// TIA Portal V20 export
FUNCTION_BLOCK "FB_PowerOn"   // FB462, SCL
{ S7_Optimized_Access := 'TRUE' }
// stored: AutoNumber false, MemoryReserve 100, SetENOAutomatically false
   VAR
      sMachinePower : Bool;
      sMachineReadySoft : Bool;
      sOkForPowerON : Bool;
      sTimeMachineReadyDelay { S7_SetPoint := 'True'} : TON_TIME;
      sDelayPowerOFF { S7_SetPoint := 'True'} : TON_TIME;
      sDelayPowerON_1 { S7_SetPoint := 'True'} : TON_TIME;
      sDelayPowerON_2 { S7_SetPoint := 'True'} : TON_TIME;
      sX_AxisBrakeRelease { S7_SetPoint := 'True'} : Bool;
      sY_AxisBrakeRelease : Bool;
      sB_AxisBrakeRelease : Bool;
   END_VAR
   VAR CONSTANT
      TIME_MACHINE_IN_DELAY : Time := T#2S;   // Output short pulse blinking
   END_VAR
BEGIN
   REGION Description header 
       //==================================================================================
       // POSALUX Swiss SA / (C) Copyright 2024
       //----------------------------------------------------------------------------------
       // Title: Power de la machine
       // Comment/Function: 
       //  A revoir le power des differents elements
       // Author: Gowsigan SRITHARAN
       // Engineering: TIA Portal v17
       //----------------------------------------------------------------------------------
       // Change log table:
       // Version  | Date     | Expert in charge | Changes applied
       // ---------|----------|------------------|------------------------------------
       // 00.00.01 | 20241120 | GSR              | First released version
       // ==================================================================================
   END_REGION

   REGION General Circuit breaker
       IF NOT "DB_DigitalInputs".sBreakerCtrl.sSWStatus THEN
           "LBP_AlarmMsgs".UserA[0].A70UUxx[3] := TRUE;
       END_IF;
   END_REGION

   REGION Operating counter
       "DB_DigitalOutputs".sOperatingCounter.sSWStatus :=
       ("LBP_Chan1".E_ProgRunning
       OR "LBP_Chan1".E_ProgWait)
       AND "LBP_ModeGroup".E_AUTO;
   END_REGION

   REGION Axis power requested
       #sOkForPowerON := "LBP_NC".E_NCKready AND "LBP_NC".E_DrivesInCylOp AND "DB_DataFromSafety".EmergencyStop AND NOT "DB_Alarms".sAlarmsLevel5 AND NOT "DB_Alarms".sAlarmsLevel6;

       IF #sOkForPowerON AND "DB_McpKeyboardSignals".sPowerON.sKeySWPositiveFront THEN
           #sMachinePower := TRUE;
       END_IF;

       IF  "DB_McpKeyboardSignals".sPowerOFF.sKeySWNegativeFront
           OR "DB_Machineshutdown_UPS".sShutDownPower
           OR "DB_Alarms".sAlarmsLevel5
           OR NOT "DB_DataFromSafety".EmergencyStop THEN
           #sMachinePower := FALSE;
       END_IF;

   END_REGION

   REGION Axis power output and waiting machine ready
       #sDelayPowerOFF(IN := NOT "LBP_NC".E_611Dready AND NOT #sMachinePower,
                       PT := T#1s);

       #sDelayPowerON_1(IN := "DB_DigitalOutputs".sInfeedON.sSWStatus,
                        PT := t#2s);
       #sDelayPowerON_2(IN := "DB_DigitalOutputs".sAxisActivation.sSWStatus,
                        PT := t#2s);
       IF #sMachinePower THEN
           "DB_DigitalOutputs".sInfeedON.sSWStatus := TRUE;
           IF #sDelayPowerON_1.Q THEN
               "DB_DigitalOutputs".sAxisActivation.sSWStatus := TRUE;
           END_IF;
           IF #sDelayPowerON_2.Q THEN

               "DB_DigitalOutputs".sAxis2_PowerContactor.sSWStatus  := TRUE;
               "DB_DigitalOutputs".sXY_AxisPowerContactor.sSWStatus := TRUE;
               "DB_DigitalOutputs".sBus60V_PowerContactor.sSWStatus := TRUE;
           END_IF;
       ELSE
           "DB_DigitalOutputs".sAxisActivation.sSWStatus := FALSE;

           IF #sDelayPowerOFF.Q THEN
               "DB_DigitalOutputs".sAxis2_PowerContactor.sSWStatus  := FALSE;
               "DB_DigitalOutputs".sXY_AxisPowerContactor.sSWStatus := FALSE;
               "DB_DigitalOutputs".sBus60V_PowerContactor.sSWStatus := FALSE;
               "DB_DigitalOutputs".sInfeedON.sSWStatus := FALSE;
           END_IF;
       END_IF;

       #sMachineReadySoft := "LBP_NC".E_611Dready;
   END_REGION

   REGION Machine in delay
       #sTimeMachineReadyDelay.TON(IN := #sMachineReadySoft,
                                   PT := #TIME_MACHINE_IN_DELAY);
   END_REGION

   REGION LED Machine ready start
       "DB_McpKeyboardSignals".sPowerON.sLedSWStatus :=
       (NOT #sMachinePower AND #sOkForPowerON AND "Clock_0.5Hz")
       OR (NOT #sTimeMachineReadyDelay.Q AND #sMachinePower AND "Clock_2Hz")
       OR #sTimeMachineReadyDelay.Q AND #sMachineReadySoft;
   END_REGION

   REGION Axis Brake
       // X Axis Brake Activation
       "DB_DigitalOutputs".sX_AxisBrakeActivation.sSWStatus := (("LBP_Axis01_X".E_AxisReady
       AND "LBP_Axis01_X".E_MotOK
       AND "LBP_Axis01_X".E_PulseEnable)
       OR #sX_AxisBrakeRelease);

       // Y Axis Brake Activation    
       "DB_DigitalOutputs".sY_AxisBrakeActivation.sSWStatus := (("LBP_Axis02_Y".E_AxisReady
       AND "LBP_Axis02_Y".E_MotOK
       AND "LBP_Axis02_Y".E_PulseEnable)
       OR #sY_AxisBrakeRelease);

       // B Axis Brake Activation   
       "DB_DigitalOutputs".sB_AxisBrakeRelease.sSWStatus := ("LBP_Axis04_B".E_AxisReady
       AND "LBP_Axis05_U1".E_MotOK
       AND "LBP_Axis05_U1".E_PulseEnable)
       OR #sB_AxisBrakeRelease;

       // Axis feed stop
       "LBP_AlarmMsgs".AxisA[1].AAFdStop60AAxx[0] := NOT "DB_DigitalOutputs".sX_AxisBrakeActivation.sSWStatus;     // X Axis
       "LBP_AlarmMsgs".AxisA[2].AAFdStop60AAxx[0] := NOT "DB_DigitalOutputs".sY_AxisBrakeActivation.sSWStatus;     // Y Axis
       "LBP_AlarmMsgs".AxisA[4].AAFdStop60AAxx[0] := NOT "DB_DigitalOutputs".sB_AxisBrakeRelease.sSWStatus;        // B Axis
   END_REGION
END_FUNCTION_BLOCK
